PROGRAM main
VAR_OUTPUT
    S1_LiDAR_Posisi AT %QX0.1 : BOOL; (* TRUE jika LiDAR mendeteksi posisi truk sudah pas/pas di tengah. *)
    S2_LoadCell_Stable AT %QX0.2 : BOOL; (* TRUE jika pembacaan berat dari load cell sudah stabil (tidak fluktuatif). *)
    Reset_Button AT %QX0.3 : BOOL; (* Tombol untuk meriset sistem setelah truk selesai ditimbang dan keluar. *)
    PC_ANPR_Truk_Detected AT %QX0.0 : BOOL; (* Diaktifkan oleh PC (Kamera) via Modbus jika plat nomor sukses terbaca. menggantikan S0_Truk_Masuk. *)
  END_VAR
  VAR
    LiDAR_Volume_Raw AT %QW20 : UINT; (* Data raw volume dari LiDAR. *)
    LoadCell_Weight_Raw AT %QW21 : UINT; (* Data raw berat dari Load Cell. *)
    Database_Tare_Weight AT %QW22 : UINT; (* Data berat kosong truk yang dikirim oleh PC dari database. *)
    Sistem_Ready : BOOL; (* Lampu indikator jembatan timbang siap menerima truk. *)
    Alarm_Posisi AT %QX0.6 : BOOL; (* Lampu/sirine jika truk berhenti di posisi yang salah. *)
    Density_Result AT %QW31 : UINT; (* Hasil akhir perhitungan massa jenis (p). *)
    Netto_Weight AT %QW30 : UINT; (* Hasil pengurangan berat total dengan berat kosong dari database. *)
    Palang_masuk AT %QX0.4 : BOOL; (* palang fisik pengontrol antrian *)
    Lock_Data AT %QX0.7 : BOOL; (* Relay internal untuk mengunci proses kalkulasi. *)
    Volume_Locked : UINT; (* Memori untuk menyimpan data volume yang sudah dikunci. *)
    Weight_Locked : UINT; (* Memori untuk menyimpan data berat yang sudah dikunci. *)
  END_VAR

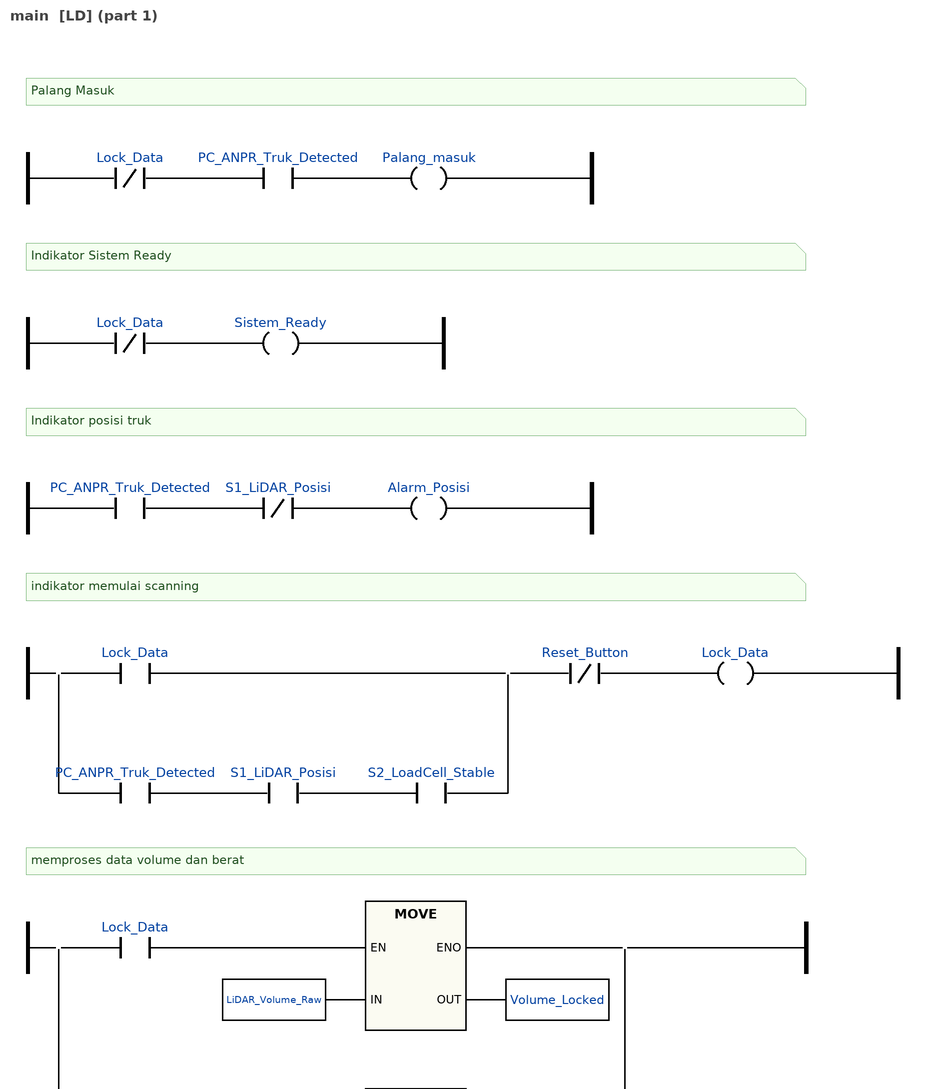
(* LD diagram, written out as Structured Text *)
(* Palang Masuk *)
Palang_masuk := NOT Lock_Data AND PC_ANPR_Truk_Detected;
(* Indikator Sistem Ready *)
Sistem_Ready := NOT Lock_Data;
(* Indikator posisi truk *)
Alarm_Posisi := PC_ANPR_Truk_Detected AND NOT S1_LiDAR_Posisi;
(* indikator memulai scanning *)
Lock_Data := (Lock_Data OR PC_ANPR_Truk_Detected AND S1_LiDAR_Posisi AND S2_LoadCell_Stable) AND NOT Reset_Button;
(* memproses data volume dan berat *)
IF Lock_Data THEN Volume_Locked := LiDAR_Volume_Raw; END_IF;
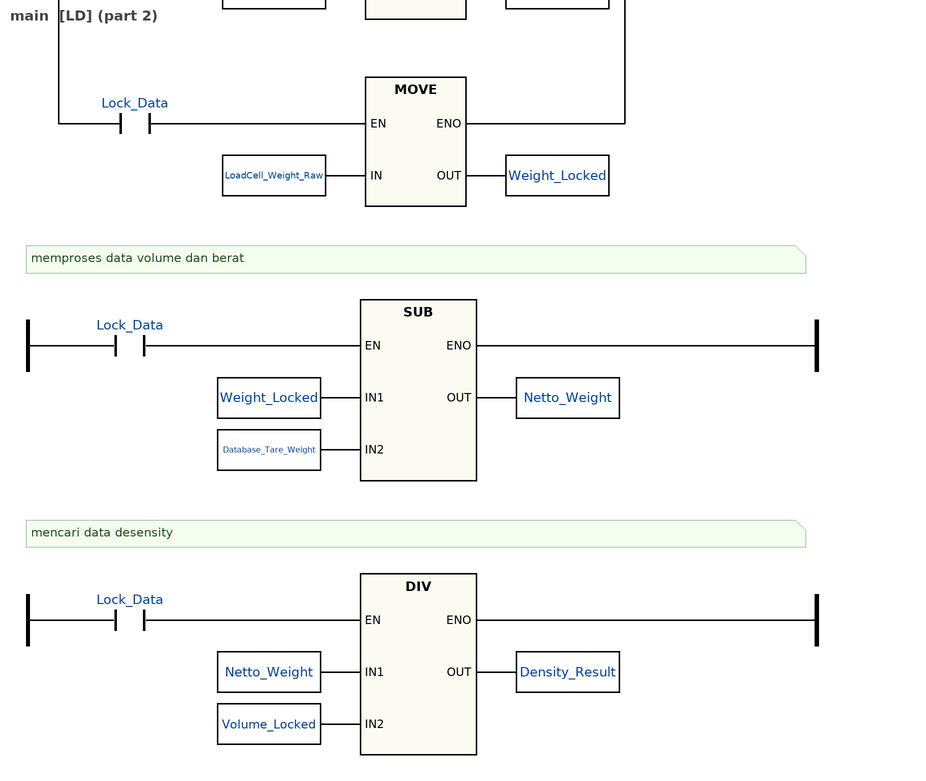
IF Lock_Data THEN Weight_Locked := LoadCell_Weight_Raw; END_IF;
(* memproses data volume dan berat *)
IF Lock_Data THEN Netto_Weight := Weight_Locked - Database_Tare_Weight; END_IF;
(* mencari data desensity *)
IF Lock_Data THEN Density_Result := Netto_Weight / Volume_Locked; END_IF;
END_PROGRAM
